// TIA Portal V18 export
TYPE "UDT_HWAlarmEntry"
// stored: IsFailsafeCompliant false
   STRUCT
      TimeStamp : DTL;   // дата/час
      SourceName : String[40];   // ім’я джерела (CPU/модуль/станція)
      Slot : UInt;   // слот (за наявності)
      Subslot : UInt;   // підслот (за наявності)
      EventID : Word;   // код події (ідентифікатор)
      ClassDiag : Bool;   // це діагностика пристрою (true)
      Appeared : Bool;   // TRUE = з’явилась, FALSE = зникла
      AckRequired : Bool;   // чи потребує ACK
      Text : String[120];   // текст події (якщо доступний)
   END_STRUCT;
END_TYPE
